PROGRAM Dummy
VAR
END_VAR

END_PROGRAM

(* stored: Version 1.1.0.1, ProductVersion 3.1.4024.12
   POU Dummy: Id {f652e54c-ae20-4eed-8a72-16ac1274cc89}, SpecialFunc None *)
